Fanuc KAREL source: kf00115.KL

-- PROVISIONAL review KL for V940-1; original PC SHA256 2b2e405dd889a51b031c57c87c9c29b98647b047d03d4b4f8263e014b60f8002
-- Incomplete behavior may be omitted. Consult companion uncertainty JSON. Do not deploy.
PROGRAM KF00115
%NOLOCKGROUP
BEGIN
  -- V9_ZERO_TABLE_METADATA_HINT layout=0001; no indexed target words; source/name/runtime held
  -- UNRESOLVED_PC offsets 0-1; opcodes 7B
  -- UNRESOLVED_PC offsets 6-18; opcodes 2D,9D,52,7F
  -- UNRESOLVED_PC offsets 23-27; opcodes 7F
  -- UNRESOLVED_PC offsets 32-48; opcodes 27,27,2E,AA,23
  -- UNRESOLVED_PC offsets 53-57; opcodes 7F
END KF00115
